// Brief: Master Arm Initialization
FUNCTION_BLOCK PUBLIC FB_ArmHome EXTENDS FB_MasterArmCtrlBase
VAR_INPUT
END_VAR
VAR_OUTPUT
END_VAR
VAR
	m_homePlanner : FB_TrajMoveJ;
	
END_VAR

// override this function in each exact controller
METHOD PROTECTED calcCmdJntPos : BOOL
VAR_INPUT
	monitorAngle :LREAL;
	slaveIdx :INT;
END_VAR

VAR_IN_OUT CONSTANT
	i_masterArm :FB_MasterArm;
	i_slaveStatus :ST_SlaveStatus;
END_VAR
VAR 
	i :INT;
	curJntVel :Vec7d;
END_VAR
// check if planner is ready
IF m_homePlanner.isGene = FALSE THEN
	calcCmdJntPos:=FALSE;
	RETURN;
END_IF

// traj plan
calcCmdJntPos :=m_homePlanner.evaluate(m_timePeriod, m_cmdJntPos,m_cmdJntVel, m_cmdJntAcc);

// check if to terminate
curJntVel :=i_masterArm.curJntVel;
m_isFinished :=m_timePeriod > m_homePlanner.duration  AND normVec7(curJntVel)<7*g_jntStaticVelThres;
END_METHOD

// override this function in each exact controller
// NOTICE: set joint control mode here, and do some initialization if needed
METHOD PROTECTED Init : BOOL
VAR_IN_OUT CONSTANT
	i_masterArm :FB_MasterArm;
	i_masterArmCtrlCmd :ST_ArmCtrlCmds;
END_VAR
VAR
	i,j :INT;
	homePosture:ARRAY[1..2] OF Vec7d;
	startJntPos,endJntPos :Vec7d;
END_VAR
SUPER^.Init(i_masterArm,i_masterArmCtrlCmd);

// traj plan
startJntPos:=i_masterArm.curJntPos;
FOR j:=1 TO 7 DO 
endJntPos[j]:=g_homePosture[i_masterArm.armIdx,j];
END_FOR
m_homePlanner.init(startJntPos,endJntPos,g_homeMaxjntVel,g_homeMaxjntAcc,g_homeMaxjntJerk);

// disable all joints
m_jntEnableFlag :=g_zeroVec7i;
m_jntEnableFlag[5]:=1;
m_jntEnableFlag[6]:=1;
m_jntEnableFlag[7]:=1;
END_METHOD

END_FUNCTION_BLOCK

(* stored: Version 1.1.0.1, ProductVersion 3.1.4024.12
   POU FB_ArmHome: Id {ff8ccb3f-4929-4315-b540-e9546f2dbd07}, SpecialFunc None
   Method calcCmdJntPos: Id {ffa3dbdd-63a1-4101-8d26-d1f3e6e5e2be}
   Method Init: Id {c6523e12-84cb-49f8-843e-9a168bb4ce28} *)
